Universal Robots PolyScope program: mojo_socket.urp

ProgramRoot setBeforeStartSequence=true; directory=/programs/usbdisk; kinematics=(a=[0, -0.425, -0.39225, 0, 0, 0], d=[0.08916, 0, 0, 0.10915, 0.09465, 0.0823], alpha=[1.5708, 0, 0, 1.5708, -1.5708, 0], deltaTheta=[0, 0, 0, 0, 0, 0], status=notInitialized); name=mojo_socket; programVersion=(project__name=PolyScope, major__version=1, minor__version=8, svn__revision=11657, build__date=Oct 09 2013, 20:14:19); robotEnvironmentFileName=default; serialNumberRobot=2013211734
  BeforeStart description=COMMAND_SEQUENCE_BEFORE_PROGRAM_START; name=BeforeStart
    Script type=1; cachedFileContents=socket_close("gripper_socket")
      | sleep(2)
      | socket_open("127.0.0.1",63352,"gripper_socket"); scriptFile=/programs/robotiq_2f_gripper_programs/rq_before_start.script
    Script type=1; cachedFileContents=###############################################################
      | # Script file used to communicate with Robotiq's gripper driver
      | # Version: DCU-1.0.10
      | ###############################################################
      | 
      | #aliases for the gripper variable names
      | ACT = 1
      | GTO = 2
      | ATR = 3
      | ARD = 4
      | FOR = 5
      | SPE = 6
      | OBJ = 7
      | STA = 8
      | FLT = 9
      | POS = 10
      | 
      | def rq_activate():
      | 	rq_gripper_act = 0
      | 	rq_set_var(ACT,1)
      | end
      | 
      | def rq_activate_and_wait():
      | 	rq_activate()
      | 
      | 	while(not rq_is_gripper_activated()):
      | 		# wait for activation completed
      | 	end
      | end
      | 
      | def rq_stop():
      | 	rq_set_var(GTO,0)
      | end
      | 
      | def rq_reset():
      | 	rq_gripper_act = 0
      | 	rq_obj_detect = 0
      | 	rq_mov_complete = 0
      | 
      | 	rq_set_var(ACT,0)
      | end
      | 
      | def rq_auto_release_open_and_wait():
      | 
      | 	rq_set_var(ARD,0)
      | 	rq_set_var(ACT,1)
      | 	rq_set_var(ATR,1)
      | 
      | 	gFLT = rq_get_var(FLT, 2)
      | 
      | 	while(not is_FLT_autorelease_completed(gFLT)):
      | 		gFLT = rq_get_var(FLT, 2)
      | 	end
      | end
      | 
      | def rq_auto_release_close_and_wait():
      | 	rq_set_var(ARD,1)
      | 	rq_set_var(ACT,1)
      | 	rq_set_var(ATR,1)
      | 
      | 	gFLT = rq_get_var(FLT, 2)
      | 
      | 	while(not is_FLT_autorelease_completed(gFLT)):
      | 		gFLT = rq_get_var(FLT, 2)
      | 	end
      | end
      | 
      | def rq_set_force(force):
      | 	rq_set_var(FOR,force)
      | end
      | 
      | def rq_set_speed(speed):
      | 	rq_set_var(SPE,speed)
      | end
      | 
      | def rq_open():
      | 	rq_move(0)
      | end
      | 
      | def rq_close():
      | 	rq_move(255)
      | end
      | 
      | def rq_open_and_wait():
      | 	rq_move_and_wait(0)
      | end
      | 
      | def rq_close_and_wait():
      | 	rq_move_and_wait(255)
      | end
      | 
      | def rq_move(pos):
      | 	rq_mov_complete = 0
      | 	rq_obj_detect = 0
      | 
      | 	rq_set_var(GTO,1)
      | 
      | 	rq_set_var(POS,pos)
      | end
      | 
      | def rq_move_and_wait(pos):
      | 	rq_move(pos)
      | 
      | 	while (not rq_is_motion_complete()):
      | 		# wait for motion completed
      | 		sleep(0.01)
      | 		sync()
      | 	end
      | 
      | 	# following code used for compatibility with previous versions
      | 	rq_is_object_detected() 
      | 
      | 	if (rq_obj_detect != 1):
      | 		rq_mov_complete = 1
      | 	end
      | end
      | 
      | def rq_is_motion_complete():
      | 	rq_mov_complete = 0
      | 
      | 	gOBJ = rq_get_var(OBJ, 1)
      | 	sleep(0.01)
      | 
      | 	if (is_OBJ_gripper_at_position(gOBJ)):
      | 		rq_mov_complete = 1
      | 		return True
      | 	end
      | 
      | 	if (is_OBJ_object_detected(gOBJ)):
      | 		rq_mov_complete = 1
      | 		return True
      | 	end
      | 
      | 	return False
      | 
      | end
      | 
      | def rq_is_gripper_activated():
      | 	gSTA = rq_get_var(STA, 1)
      | 
      | 	if(is_STA_gripper_activated(gSTA)):
      | 		rq_gripper_act = 1
      | 		return True
      | 	else:
      | 		rq_gripper_act = 0
      | 		return False
      | 	end
      | end
      | 
      | def rq_is_object_detected():
      | 	gOBJ = rq_get_var(OBJ, 1)
      | 
      | 	if(is_OBJ_object_detected(gOBJ)):
      | 		rq_obj_detect = 1
      | 		return True
      | 	else:
      | 		rq_obj_detect = 0
      | 		return False
      | 	end
      | end
      | 
      | def rq_print_fault_code():
      | 	gFLT = rq_get_var(FLT, 2)
      | 
      | 	if(is_FLT_no_fault(gFLT)):
      | 		textmsg("Gripper Fault : ", "No Fault (0x00)")
      | 	elif (is_FLT_action_delayed(gFLT)):
      | 		textmsg("Gripper Fault : ", "Priority Fault: Action delayed, initialization must be completed prior to action (0x05)")
      | 	elif (is_FLT_not_activated(gFLT)):
      | 		textmsg("Gripper Fault : ", "Priority Fault: The activation must be set prior to action (0x07)")
      | 	elif (is_FLT_autorelease_in_progress(gFLT)):
      | 		textmsg("Gripper Fault : ", "Minor Fault: Automatic release in progress (0x0B)")
      | 	elif (is_FLT_overcurrent(gFLT)):
      | 		textmsg("Gripper Fault : ", "Minor Fault: Overcurrent protection tiggered (0x0E)")
      | 	elif (is_FLT_autorelease_completed(gFLT)):
      | 		textmsg("Gripper Fault : ", "Major Fault: Automatic release completed (0x0F)")
      | 	else:
      | 		textmsg("Gripper Fault : ", "Unkwown Fault")
      | 	end
      | end
      | 
      | def rq_print_num_cycles():
      | 	socket_send_string("GET NCY","gripper_socket")
      | 	sync()
      | 	string_from_server = socket_read_string("gripper_socket")
      | 	sync()
      | 
      | 	if(string_from_server == "0"):
      | 		textmsg("Gripper Cycle Number : ", "Number of cycles is unreachable.")
      | 	else:
      | 		textmsg("Gripper Cycle Number : ", string_from_server)
      | 	end
      | end
      | 
      | def rq_print_driver_state():
      | 	socket_send_string("GET DST","gripper_socket")
      | 	sync()
      | 	string_from_server = socket_read_string("gripper_socket")
      | 	sync()
      | 
      | 	if(string_from_server == "0"):
      | 		textmsg("Gripper Driver State : ", "RQ_STATE_INIT")
      | 	elif(string_from_server == "1"):
      | 		textmsg("Gripper Driver State : ", "RQ_STATE_LISTEN")
      | 	elif(string_from_server == "2"):
      | 		textmsg("Gripper Driver State : ", "RQ_STATE_READ_INFO")
      | 	elif(string_from_server == "3"):
      | 		textmsg("Gripper Driver State : ", "RQ_STATE_ACTIVATION")
      | 	else:
      | 		textmsg("Gripper Driver State : ", "RQ_STATE_RUN")
      | 	end
      | end
      | 
      | def rq_print_serial_number():
      | 	#socket_send_string("GET SNU","gripper_socket")
      | 	#sync()
      | 	#string_from_server = socket_read_string("gripper_socket")
      | 	#sync()
      | 	#textmsg("Gripper Serial Number : ", string_from_server)
      | end
      | 
      | def rq_print_firmware_version():
      | 	socket_send_string("GET FWV","gripper_socket")
      | 	sync()
      | 	string_from_server = socket_read_string("gripper_socket")
      | 	sync()
      | 	textmsg("Gripper Firmware Version : ", string_from_server)
      | end
      | 
      | def rq_print_driver_version():
      | 	socket_send_string("GET VER","gripper_socket")
      | 	sync()
      | 	string_from_server = socket_read_string("gripper_socket")
      | 	sync()
      | 	textmsg("Gripper Driver Version : ", string_from_server)
      | end
      | 
      | def rq_print_probleme_connection():
      | 	socket_send_string("GET PCO","gripper_socket")
      | 	sync()
      | 	string_from_server = socket_read_string("gripper_socket")
      | 	sync()
      | 	if (string_from_server == "0"):
      | 		textmsg("Gripper Connection State : ", "No connection problem detected")
      | 	else:
      | 		textmsg("Gripper Connection State : ", "Connection problem detected")
      | 	end
      | end
      | 
      | def rq_current_pos():
      | 	rq_pos = socket_get_var("POS","gripper_socket")
      | 	sync()
      | end
      | 
      | # Returns True if list_of_bytes is [3, 'a', 'c', 'k']
      | def is_ack(list_of_bytes):
      | 	
      | 	# list length is not 3
      | 	if (list_of_bytes[0] != 3):
      | 		return False
      | 	end
      | 
      | 	# first byte not is 'a'?
      | 	if (list_of_bytes[1] != 97):
      | 		return False
      | 	end
      | 	
      | 	# first byte not is 'c'?
      | 	if (list_of_bytes[2] != 99):
      | 		return False
      | 	end
      | 	
      | 	# first byte not is 'k'?
      | 	if (list_of_bytes[3] != 107):
      | 		return False
      | 	end
      | 	
      | 	return True
      | end
      | 
      | # Returns True if list_of_bytes is not [3, 'a', 'c', 'k']
      | def is_not_ack(list_of_bytes):
      | 	if (is_ack(list_of_bytes)):
      | 		return False
      | 	else:
      | 		return True
      | 	end
      | end
      | 
      | def is_STA_gripper_activated (list_of_bytes):
      | 
      | 	# list length is not 1
      | 	if (list_of_bytes[0] != 1):
      | 		return False
      | 	end
      | 
      | 	# byte is '3'?
      | 	if (list_of_bytes[1] == 51):
      | 		return True
      | 	end
      | 
      | 	return False
      | end
      | 
      | # Returns True if list_of_byte is [1, '1'] or [1, '2']
      | # Used to test OBJ = 0x1 or OBJ = 0x2
      | def is_OBJ_object_detected (list_of_bytes):
      | 	
      | 	# list length is not 1
      | 	if (list_of_bytes[0] != 1):
      | 		return False
      | 	end
      | 
      | 	# byte is '2'?
      | 	if (list_of_bytes[1] == 50):
      | 		return True
      | 	end
      | 
      | 	# byte is '1'?
      | 	if (list_of_bytes[1]  == 49):
      | 		return True
      | 	end
      | 
      | 	return False
      | 	
      | end
      | 
      | # Returns True if list_of_byte is [1, '3']
      | # Used to test OBJ = 0x3
      | def is_OBJ_gripper_at_position (list_of_bytes):
      | 
      | 	# list length is not 1
      | 	if (list_of_bytes[0] != 1):
      | 		return False
      | 	end
      | 
      | 	# byte is '3'?
      | 	if (list_of_bytes[1] == 51):
      | 		return True
      | 	end
      | 	
      | 	return False
      | end
      | 
      | def is_not_OBJ_gripper_at_position (list_of_bytes):
      | 	
      | 	if (is_OBJ_gripper_at_position(list_of_bytes)):
      | 		return False
      | 	else:
      | 		return True
      | 	end
      | end
      | 
      | def is_FLT_no_fault(list_of_bytes):
      | 
      | 	# list length is not 2
      | 	if (list_of_bytes[0] != 2):
      | 		return False
      | 	end
      | 
      | 	# first byte is '0'?
      | 	if (list_of_bytes[1] != 48):
      | 		return False
      | 	end
      | 
      | 	# second byte is '0'?
      | 	if (list_of_bytes[2] != 48):
      | 		return False
      | 	end
      | 
      | 	return True
      | 
      | end
      | 
      | def is_FLT_action_delayed(list_of_bytes):
      | 
      | 	# list length is not 2
      | 	if (list_of_bytes[0] != 2):
      | 		return False
      | 	end
      | 
      | 	# first byte is '0'?
      | 	if (list_of_bytes[1] != 48):
      | 		return False
      | 	end
      | 
      | 	# second byte is '5'?
      | 	if (list_of_bytes[2] != 53):
      | 		return False
      | 	end
      | 
      | 	return True
      | end
      | 
      | def is_FLT_not_activated(list_of_bytes):
      | 
      | 	# list length is not 2
      | 	if (list_of_bytes[0] != 2):
      | 		return False
      | 	end
      | 
      | 	# first byte is '0'?
      | 	if (list_of_bytes[1] != 48):
      | 		return False
      | 	end
      | 
      | 	# second byte is '7'?
      | 	if (list_of_bytes[2] != 55):
      | 		return False
      | 	end
      | 
      | 	return True
      | end
      | 
      | def is_FLT_autorelease_in_progress(list_of_bytes):
      | 
      | 	# list length is not 2
      | 	if (list_of_bytes[0] != 2):
      | 		return False
      | 	end
      | 
      | 	# first byte is '1'?
      | 	if (list_of_bytes[1] != 49):
      | 		return False
      | 	end
      | 
      | 	# second byte is '1'?
      | 	if (list_of_bytes[2] != 49):
      | 		return False
      | 	end
      | 
      | 	return True
      | 
      | end
      | 
      | def is_FLT_overcurrent(list_of_bytes):
      | 
      | 	# list length is not 2
      | 	if (list_of_bytes[0] != 2):
      | 		return False
      | 	end
      | 
      | 	# first byte is '1'?
      | 	if (list_of_bytes[1] != 49):
      | 		return False
      | 	end
      | 
      | 	# second byte is '4'?
      | 	if (list_of_bytes[2] != 52):
      | 		return False
      | 	end
      | 
      | 	return True
      | 
      | end
      | 
      | def is_FLT_autorelease_completed(list_of_bytes):
      | 
      | 	# list length is not 2
      | 	if (list_of_bytes[0] != 2):
      | 		return False
      | 	end
      | 
      | 	# first byte is '1'?
      | 	if (list_of_bytes[1] != 49):
      | 		return False
      | 	end
      | 
      | 	# second byte is '5'?
      | 	if (list_of_bytes[2] != 53):
      | 		return False
      | 	end
      | 
      | 	return True
      | 
      | end
      | 
      | def rq_set_var(var_id, var_value):
      | 	
      | 	var_name = ""
      | 
      | 	sync()
      | 	if   (var_id == ACT):
      | 		var_name = "ACT"
      | 	elif (var_id == GTO):
      | 		var_name = "GTO"
      | 	elif (var_id == ATR):
      | 		var_name = "ATR"
      | 	elif (var_id == ARD):
      | 		var_name = "ARD"
      | 	elif (var_id == FOR):
      | 		var_name = "FOR"
      | 	elif (var_id == SPE):
      | 		var_name = "SPE"
      | 	elif (var_id == POS):
      | 		var_name = "POS"
      | 	else:
      | 	end
      | 
      | 	socket_set_var(var_name, var_value, "gripper_socket")
      | 	sync()
      | 	ack = socket_read_byte_list(3, "gripper_socket")
      | 	sync()
      | 
      | 	while(is_not_ack(ack)):
      | 
      | 		textmsg("rq_set_var : retry", " ...")
      | 		textmsg("rq_set_var : var_name = ", var_name)
      | 		textmsg("rq_set_var : var_value = ", var_value)
      | 
      | 		if (ack[0] != 0):
      | 			textmsg("rq_set_var : invalid ack value = ", ack)
      | 		end
      | 
      | 		socket_set_var(var_name , var_value,"gripper_socket")
      | 		sync()
      | 		ack = socket_read_byte_list(3, "gripper_socket")
      | 		sync()
      | 	end
      | end
      | 
      | 
      | def rq_get_var(var_name, nbr_bytes):
      | 	
      | 	if (var_name == FLT):
      | 		socket_send_string("GET FLT","gripper_socket")
      | 		sync()
      | 	elif (var_name == OBJ):
      | 		socket_send_string("GET OBJ","gripper_socket")
      | 		sync()
      | 	elif (var_name == STA):
      | 		socket_send_string("GET STA","gripper_socket")
      | 		sync()
      | 	else:
      | 	end
      | 	
      | 	var_value = socket_read_byte_list(nbr_bytes, "gripper_socket")
      | 	sync()
      | 
      | 	return var_value
      | end; scriptFile=/programs/robotiq_2f_gripper_programs/rq_script.script
    Assignment assignmentValueSource=0; expr=0; operatorValueType=INTEGER; valueSource=EXPRESSION; variable=0
    Assignment assignmentValueSource=0; expr=0; operatorValueType=INTEGER; valueSource=EXPRESSION; variable=0
    Assignment assignmentValueSource=0; expr=255; operatorValueType=INTEGER; valueSource=EXPRESSION; variable=0
    CallSubProgram subProgramNodeToCall=rq_set_force(rq_force)
    CallSubProgram subProgramNodeToCall=rq_set_speed(rq_speed)
    CallSubProgram subProgramNodeToCall=rq_activate_and_wait()
    CallSubProgram subProgramNodeToCall=rq_open_and_wait()
    Assignment assignmentValueSource=0; expr=[6,0,0,0,0,0,0]; operatorValueType=INTEGER; valueSource=EXPRESSION; variable=(name=receive_data, prefersPersistentValue=false, requestANewUniqueName=false)
    Assignment assignmentValueSource=0; expr=[0,-1.5708,0,-1.5708,0,0]; operatorValueType=INTEGER; valueSource=EXPRESSION; variable=(name=Move_To_Joints, prefersPersistentValue=false, requestANewUniqueName=false)
    Suppressed suppressedNode=p[0.100,-0.175,0.700,-1.2,2.5,-0.8]
    Assignment assignmentValueSource=0; expr=get_target_tcp_pose(); operatorValueType=INTEGER; valueSource=EXPRESSION; variable=(name=Move_To_Tcp, prefersPersistentValue=false, requestANewUniqueName=false)
    Assignment assignmentValueSource=0; expr=[0]; operatorValueType=INTEGER; valueSource=EXPRESSION; variable=(name=Move_To_Gripper, prefersPersistentValue=false, requestANewUniqueName=false)
    CallSubProgram subProgramNodeToCall=pose_1=get_joint_positions()
    Script type=0; expressionBranchNode=socket_close("robot_socket")
    Script type=0; expressionBranchNode=sleep(2)
    Script type=0; expressionBranchNode=socket_open("172.31.1.21",30000,"robot_socket")
    Assignment assignmentValueSource=0; expr=[0,0]; operatorValueType=INTEGER; valueSource=EXPRESSION; variable=(name=task, prefersPersistentValue=false, requestANewUniqueName=false)
    Assignment assignmentValueSource=0; expr=0; operatorValueType=INTEGER; valueSource=EXPRESSION; variable=(name=coop, prefersPersistentValue=false, requestANewUniqueName=false)
    Assignment assignmentValueSource=0; expr=False; operatorValueType=INTEGER; valueSource=EXPRESSION; variable=(name=tcp_ctrl, prefersPersistentValue=false, requestANewUniqueName=false)
  MainProgram cartesianAcceleration=1.2; cartesianSpeed=0.25; jointAcceleration=1.3962634015954636; jointSpeed=1.0471975511965976; moveAsFastAsPossible=true; sharedProcessMoveBlendRadius=0.025; featureReference=(installationNameReference=Base); motionType=JOINT_SPACE
    Suppressed suppressedNode=___tran51ate_this_name___Joint_0_name
    Suppressed suppressedNode=1
    Suppressed 
    Suppressed suppressedNode=0
    Script type=0; expressionBranchNode=ExpressionVariableNode=socket_read_ascii_float(1,"robot_socket")
    If expr=ExpressionVariableNode[1]≟2; type=IF_NODE
      CallSubProgram subProgramNodeToCall=pose_1=get_joint_positions()
      Assignment assignmentValueSource=0; expr=[0,0]; operatorValueType=INTEGER; valueSource=EXPRESSION; variable=(name=task, prefersPersistentValue=false, requestANewUniqueName=false)
    If expr=task[1]≟3; type=ELSEIF_NODE
      CallSubProgram subProgramNodeToCall=rq_open_and_wait()
      Script type=0; expressionBranchNode=socket_send_string("1","robot_socket")
      Assignment assignmentValueSource=0; expr=[0,0]; operatorValueType=INTEGER; valueSource=EXPRESSION; variable=(name=task, prefersPersistentValue=false, requestANewUniqueName=false)
    If expr=task[1]≟4; type=ELSEIF_NODE
      CallSubProgram subProgramNodeToCall=rq_close_and_wait()
      Script type=0; expressionBranchNode=socket_send_string("1","robot_socket")
      Assignment assignmentValueSource=0; expr=[0,0]; operatorValueType=INTEGER; valueSource=EXPRESSION; variable=(name=task, prefersPersistentValue=false, requestANewUniqueName=false)
    If expr=task[1]≟5; type=ELSEIF_NODE
      Script type=0; expressionBranchNode=tcp_pose=get_actual_tcp_pose()
      Script type=0; expressionBranchNode=socket_send_string(tcp_pose,"robot_socket")
      Assignment assignmentValueSource=0; expr=[0,0]; operatorValueType=INTEGER; valueSource=EXPRESSION; variable=(name=task, prefersPersistentValue=false, requestANewUniqueName=false)
    If expr=task[1]≟1; type=ELSEIF_NODE
      CallSubProgram subProgramNodeToCall=receive_data=socket_read_ascii_float(6,"robot_socket")
    If expr=task[1]≟6; type=ELSEIF_NODE
      CallSubProgram subProgramNodeToCall=receive_data=socket_read_ascii_float(6,"robot_socket")
    If expr=ExpressionVariableNode[1]≟7; type=ELSEIF_NODE
      CallSubProgram subProgramNodeToCall=receive_data=socket_read_ascii_float(1,"robot_socket")
    Wait analogComparison=0; analogInputRange=0; analogValue=0.0; digitalValue=0; selectedAnalogSensor=-1; selectedDigitalSensor=-1; waitTime=0.01; type=NO_WAIT
  Thread name=Thread_1
    If expr=coop≟1; type=IF_NODE
      While count=0; expr=coop≟1; type=LOOP_EXPR; variable=(name=Loop_3, prefersPersistentValue=false, requestANewUniqueName=false)
        Force feature__reference=(installationNameReference=Base); force__mode__wrench=[0, 0, 0, 0, 0, 0]; limits__force=[0.15, 0.15, 0.15, 1.0472, 1.0472, 1.0472]; limits__motion=[0.1, 0.1, 0.1, 0.17453, 0.17453, 0.17453]; selection__vector=[1, 1, 1, 1, 1, 1]; type=FORCE_TYPE_FRAME
          Wait analogComparison=0; analogInputRange=0; analogValue=0.0; digitalValue=0; selectedAnalogSensor=-1; selectedDigitalSensor=-1; waitTime=0.01; type=TIMER_WAIT
      Assignment assignmentValueSource=0; expr=0; operatorValueType=INTEGER; valueSource=EXPRESSION; variable=(name=coop, prefersPersistentValue=false, requestANewUniqueName=false)
      CallSubProgram subProgramNodeToCall=pose_1=get_joint_positions()
    If type=ELSE_NODE
      If expr=not ExpressionVariableNode; type=IF_NODE
        Script type=0; expressionBranchNode=movej(Move_To_Joints,a=0.2,v=0.3,r=0)
      If type=ELSE_NODE
        Script type=0; expressionBranchNode=movel(Move_To_Tcp,a=0.1,v=0.15,r=0)
      Wait analogComparison=0; analogInputRange=0; analogValue=0.0; digitalValue=0; selectedAnalogSensor=-1; selectedDigitalSensor=-1; waitTime=0.01; type=TIMER_WAIT
  Thread name=Thread_2
    Script type=0; expressionBranchNode=rq_move(Move_To_Gripper[0])
  subProgramToCall name=SubProgram_1
    Script type=0; expressionBranchNode=receive_data=socket_read_ascii_float(6,"robot_socket")
    If expr=ExpressionVariableNode[0]≠6; type=IF_NODE
      Script type=0; expressionBranchNode=socket_send_string("0","robot_socket")
    If type=ELSE_NODE
      Script type=0; expressionBranchNode=socket_send_string("1","robot_socket")
      Assignment assignmentValueSource=0; expr=0; operatorValueType=INTEGER; valueSource=EXPRESSION; variable=(name=pointer, prefersPersistentValue=false, requestANewUniqueName=false)
      While count=0; expr=ExpressionVariableNode<ExpressionVariableNode[0]; type=LOOP_EXPR; variable=(name=Loop_1, prefersPersistentValue=false, requestANewUniqueName=false)
        Script type=0; expressionBranchNode=Move_To_Joints[pointer]=receive_data[pointer+1]
        Assignment assignmentValueSource=0; expr=ExpressionVariableNode+1; operatorValueType=INTEGER; valueSource=EXPRESSION; variable=(name=pointer, prefersPersistentValue=false, requestANewUniqueName=false)
      Assignment assignmentValueSource=0; expr=[0,0]; operatorValueType=INTEGER; valueSource=EXPRESSION; variable=(name=task, prefersPersistentValue=false, requestANewUniqueName=false)
  subProgramToCall name=SubP_set_tcp
    Script type=0; expressionBranchNode=receive_data=socket_read_ascii_float(6,"robot_socket")
    If expr=ExpressionVariableNode[0]≠6; type=IF_NODE
      Script type=0; expressionBranchNode=socket_send_string("0","robot_socket")
    If type=ELSE_NODE
      Script type=0; expressionBranchNode=socket_send_string("1","robot_socket")
      Assignment assignmentValueSource=0; expr=0; operatorValueType=INTEGER; valueSource=EXPRESSION; variable=(name=pointer, prefersPersistentValue=false, requestANewUniqueName=false)
      While count=0; expr=ExpressionVariableNode<ExpressionVariableNode[0]; type=LOOP_EXPR; variable=(name=Loop_4, prefersPersistentValue=false, requestANewUniqueName=false)
        Script type=0; expressionBranchNode=Move_To_Tcp[pointer]=receive_data[pointer+1]
        Assignment assignmentValueSource=0; expr=ExpressionVariableNode+1; operatorValueType=INTEGER; valueSource=EXPRESSION; variable=(name=pointer, prefersPersistentValue=false, requestANewUniqueName=false)
      Assignment assignmentValueSource=0; expr=[0,0]; operatorValueType=INTEGER; valueSource=EXPRESSION; variable=(name=task, prefersPersistentValue=false, requestANewUniqueName=false)
  subProgramToCall name=SubP_set_grip
    Script type=0; expressionBranchNode=receive_data=socket_read_ascii_float(1,"robot_socket")
    If expr=ExpressionVariableNode[0]≠1; type=IF_NODE
      Script type=0; expressionBranchNode=socket_send_string("0","robot_socket")
    If type=ELSE_NODE
      Script type=0; expressionBranchNode=socket_send_string("1","robot_socket")
      Assignment assignmentValueSource=0; expr=0; operatorValueType=INTEGER; valueSource=EXPRESSION; variable=(name=pointer, prefersPersistentValue=false, requestANewUniqueName=false)
      While count=0; expr=ExpressionVariableNode<ExpressionVariableNode[0]; type=LOOP_EXPR; variable=(name=Loop_5, prefersPersistentValue=false, requestANewUniqueName=false)
        Script type=0; expressionBranchNode=Move_To_Gripper[pointer]=receive_data[pointer+1]
        Assignment assignmentValueSource=0; expr=ExpressionVariableNode+1; operatorValueType=INTEGER; valueSource=EXPRESSION; variable=(name=pointer, prefersPersistentValue=false, requestANewUniqueName=false)
      Assignment assignmentValueSource=0; expr=[0,0]; operatorValueType=INTEGER; valueSource=EXPRESSION; variable=(name=task, prefersPersistentValue=false, requestANewUniqueName=false)
  subProgramToCall name=SubProgram_2
    Script type=0; expressionBranchNode=pose_1=get_joint_positions()
    Script type=0; expressionBranchNode=socket_send_string(pose_1,"robot_socket")
  subProgramToCall name=SubProgram_3
    Script type=0; expressionBranchNode=pose_1=get_joint_positions()
    Assignment assignmentValueSource=0; expr=0; operatorValueType=INTEGER; valueSource=EXPRESSION; variable=(name=pointer, prefersPersistentValue=false, requestANewUniqueName=false)
    While count=0; expr=ExpressionVariableNode<ExpressionVariableNode[0]; type=LOOP_EXPR; variable=(name=Loop_2, prefersPersistentValue=false, requestANewUniqueName=false)
      Script type=0; expressionBranchNode=Move_To_Joints[pointer]=pose_1[pointer]
      Assignment assignmentValueSource=0; expr=ExpressionVariableNode+1; operatorValueType=INTEGER; valueSource=EXPRESSION; variable=(name=pointer, prefersPersistentValue=false, requestANewUniqueName=false)
  subProgramToCall [hidden by the author, left out]
  subProgramToCall [hidden by the author, left out]
  subProgramToCall [hidden by the author, left out]
  SubProgram [hidden by the author, left out]
  subProgramToCall [hidden by the author, left out]
  subProgramToCall [hidden by the author, left out]
